FUNCTION_BLOCK BadRandom
  (* Standard: 61499-2 *)
  (* Version 0.1, 2017-00-02, hpea485, UOA *)
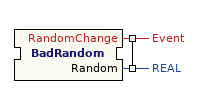
  EVENT_OUTPUT
    RandomChange WITH Random;
  END_EVENT
  VAR_OUTPUT
    Random : REAL;
  END_VAR
  VAR
    Len : INT := 10;
    Pos : INT := 0;
    Vals : ARRAY [0..9] OF REAL := [0.01,0.05,-0.02,0.03,-0.04,-0.02,0.01,0.03,-0.02,-0.02];
  END_VAR
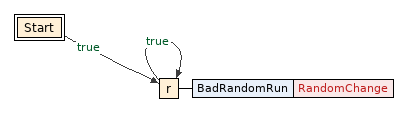
  EC_STATES
    Start;
    r : BadRandomRun -> RandomChange;
  END_STATES
  EC_TRANSITIONS
    Start TO r := true;
    r TO r := true;
  END_TRANSITIONS
  ALGORITHM BadRandomRun IN C:
me->Random = me->Vals[me->Pos];

me->Pos++;

if(me->Pos >= me->Len) {
	me->Pos = 0;
}
  END_ALGORITHM
END_FUNCTION_BLOCK
